// TIA Portal V18 export
DATA_BLOCK "Room2_SearchArea_idb"   // DB7
VERSION : 0.1
// stored: AutoNumber true, DBAccessibleFromOPCUA true, InstanceOfName SearchArea, InstanceOfType FB
"SearchArea"
   // VAR_INPUT
   //    SB1 : Bool;
   //    SB2 : Bool;
   //    Door : Bool;
   //    "E-Stop" : Bool;
   //    SearchArea_Time : Time;
   //    Reset : Bool;
   // END_VAR
   // VAR
   //    SearchArea_Timer { S7_SetPoint := 'True'} : TON_TIME;
   //    SearchArea_Status : Int;
   //    "Step" { S7_SetPoint := 'True'} : Int;
   //    Error { ExternalAccessible := 'False'; ExternalVisible := 'False'; ExternalWritable := 'False'} : Struct
   //       All { ExternalAccessible := 'False'; ExternalVisible := 'False'; ExternalWritable := 'False'} : Bool;
   //       StartFail { ExternalAccessible := 'False'; ExternalVisible := 'False'; ExternalWritable := 'False'} : Bool;
   //       WrongSequence1 { ExternalAccessible := 'False'; ExternalVisible := 'False'; ExternalWritable := 'False'} : Bool;
   //       WrongSequence2 { ExternalAccessible := 'False'; ExternalVisible := 'False'; ExternalWritable := 'False'} : Bool;
   //       Timeout { ExternalAccessible := 'False'; ExternalVisible := 'False'; ExternalWritable := 'False'} : Bool;
   //    END_STRUCT;
   // END_VAR
BEGIN
END_DATA_BLOCK
